(* PLC project Template, CODESYS CODESYS V3.5 SP17 Patch 3 *)
(* stored: creationDateTime 2026-02-13T14:33:38.6413633, version 3.5.17.30, modificationDateTime 2026-02-13T14:07:44.0721923, organization organization *)

{attribute 'qualified_only'}
{attribute 'strict'}
TYPE e_SaveReadJSONFileStates : (STATE_IDLE := 0, STATE_COMBINE, STATE_COMPOSE, STATE_SAVE, STATE_FINISH, STATE_PARSE, STATE_READ);
END_TYPE

FUNCTION_BLOCK FB_ReadJSONFile
  VAR CONSTANT
    SplitSize : INT := 1024;
  END_VAR
  VAR_INPUT
    xStart : BOOL;
    sFileName : STRING(255);
    pJSOBJ : POINTER TO ARRAY[1..GPL_JSON.MAX_VARS] OF JSONVAR;  (* pointer to local structure made up of type JSONVAR *)
    udiSize : UDINT;  (* SHOULD BE EQUAL TO SIZEOF(JSONOBJ) , *)
  END_VAR
  VAR_OUTPUT
    xBusy : BOOL;
    xDone : BOOL;
    xError : BOOL;
  END_VAR
  VAR
    state : e_SaveReadJSONFileStates := e_SaveReadJSONFileStates.STATE_IDLE;
    xStartRE : R_TRIG;
    xAutoReset : BOOL := TRUE;
    fread : FB_ReadTxtFile;
    ParseJSON : JSON_TO_STRUCT;  (* Part of PRO_JSON *)
    sContent : STRING(GPL_JSON.MAX_JSON_STRING);
    sLastError : STRING;
  END_VAR

            xStartRE(CLK:=xStart);
CASE state OF
	e_SaveReadJSONFileStates.STATE_IDLE:
		IF xStartRE.Q THEN
			state:=e_SaveReadJSONFileStates.STATE_READ;
			xDone:=FALSE;
			xBusy:=TRUE;
			xError:=FALSE;
			sLastError:='';
			sContent:='';
		END_IF

	e_SaveReadJSONFileStates.STATE_READ:
		fread(sFileName:=sFileName,
			result:=sContent,
			xStart:=TRUE);	
	
		IF fread.xDone THEN
			state:=e_SaveReadJSONFileStates.STATE_PARSE;
		END_IF
		IF fread.xError THEN
			state:=e_SaveReadJSONFileStates.STATE_FINISH;
			xError:=TRUE;
			sLastError:='File reading';
		END_IF

	e_SaveReadJSONFileStates.STATE_PARSE:
		ParseJSON(JSONString:=ADR(sContent),
				JSONStringSize:=SIZEOF(sContent),
				JSONVars:=pJSOBJ,
				NumberOfVars:=udiSIZE/SIZEOF(JSONVAR),
				Execute:=TRUE);

		IF  ParseJSON.Done THEN
			state:=e_SaveReadJSONFileStates.STATE_FINISH;
		END_IF
		IF ParseJSON.Error THEN
			state:=e_SaveReadJSONFileStates.STATE_FINISH;
			xError:=TRUE;
			sLastError:='JSON parsing';
		END_IF

	e_SaveReadJSONFileStates.STATE_FINISH:
		xBusy:=FALSE;
		xDone:=TRUE;

		IF xAutoReset THEN
			Reset();
		END_IF
		ParseJSON(Execute:=TRUE);
		state:=e_SaveReadJSONFileStates.STATE_IDLE;
END_CASE

          

METHOD Reset : BOOL
                  state:=e_SaveReadJSONFileStates.STATE_IDLE;
sContent:='';
ParseJSON(Execute:=FALSE);
ParseJSON.ClearAll();
xError:=FALSE;
Reset:=TRUE;
xStartRE(CLK:=FALSE);
                
END_METHOD
END_FUNCTION_BLOCK

{attribute 'contains_implicit_enum'}
FUNCTION_BLOCK FB_ReadTxtFile
  VAR CONSTANT
    SplitSize : INT := 1024;
  END_VAR
  VAR_INPUT
    xStart : BOOL;
    sFileName : REFERENCE TO STRING(255);
    Result : REFERENCE TO STRING(GPL_JSON.MAX_JSON_STRING);
  END_VAR
  VAR_OUTPUT
    xBusy : BOOL;
    xDone : BOOL;
    xError : BOOL;
  END_VAR
  VAR
    fopen : FILE.Open;
    fread : FILE.Read;
    fclose : FILE.Close;
    xStartRE : R_TRIG;
    xAutoReset : BOOL := TRUE;
    {attribute 'implicit_enum_type'}
    step : Implicit_Enum__FB_ReadTxtFile__step;
    tempString : STRING(GPL_JSON.MAX_JSON_STRING);
    endPos : INT;
    subString : STRING(SplitSize);  (* Not more than CLEANSTRING.MAXSTRING; *)
    cleanupCount : INT := 0;
    cleanupCounter : INT;
    tmp : REAL;
    startPos : INT;
    finishPos : INT;
    lenCopy : DINT;
    pos : INT;
    testChar : STRING(1) := '"';
    testStr : STRING(1);
  END_VAR

            xStartRE(CLK:=xStart);
CASE step OF
	STEP_IDLE:
		IF xStartRE.Q AND NOT xError THEN
			step:=STEP_OPEN;
			xDone:=FALSE;
			xBusy:=TRUE;
			xError:=FALSE;			
		END_IF
		
		fopen(xExecute:=FALSE);
    	fread(xExecute:=FALSE);
		fclose(xExecute:=FALSE);
	
	STEP_OPEN:
		fopen.sFileName:=sFileName;
		fopen.eFileMode:=FILE.MODE.MREAD;
		fopen.xExclusive:=TRUE;
		fopen(xExecute:=TRUE);
		
		IF fopen.xDone THEN
			step:=STEP_READ;
		END_IF
		IF fopen.xError THEN
			step:=STEP_CLOSE;
			xError:=TRUE;
		END_IF
		
	STEP_READ:
		Result:='';
		fread.hFile:=fopen.hFile;
		
		fread.pBuffer:=ADR(tempString);
		
		fread.szBuffer:=SIZEOF(tempString);
		fread(xExecute:=TRUE);
		IF fread.xDone THEN
			step:=STEP_CLEANUP;
			endPos:=TO_INT(StrLenA(ADR(tempString)));
			startPos:=1; 
			cleanupCounter:=0;
			
			cleanupCount:=TO_INT(endPos/SplitSize);
			//Simple Round up
			tmp:=TO_REAL(endPos)/TO_REAL(SplitSize);
			IF tmp>TO_REAL(cleanupCount) THEN
				cleanupCount:=cleanupCount+1;
			END_IF
			
		END_IF
		IF fread.xError THEN
			step:=STEP_CLOSE;
			xError:=TRUE;
		END_IF
	STEP_CLEANUP:
		
		finishPos := MIN(endPos, startPos + SplitSize - 1);
		pos:=finishPos;
		lenCopy   := finishPos - startPos + 1;  
		IF lenCopy>0 THEN
			STU.StrMidA(ADR(tempString),SIZEOF(tempString),TO_INT(lenCopy),startPos,ADR(subString),TO_UINT(SplitSize+1));
			CleanupString(); //Save spaces
			STU.StrConcatA(ADR(subString),ADR(Result),TO_INT(SIZEOF(Result)));
		END_IF
		
		IF finishPos>=endPos THEN 
			step:=STEP_CLOSE;
		END_IF
		startPos:=finishPos+1;
		cleanupCounter:=cleanupCounter+1;
		IF cleanupCounter>cleanupCount THEN 
			step:=STEP_CLOSE;
		END_IF
	STEP_CLOSE:
		fclose.hFile:=fopen.hFile;
		fclose(xExecute:=TRUE);
		IF fclose.xDone THEN
			step:=STEP_FINISH;
		END_IF
		IF fclose.xError THEN
			step:=STEP_FINISH;
			xError:=TRUE;
		END_IF
		
	STEP_FINISH:
		IF xAutoReset AND xError THEN
			Reset();
		END_IF
		step:=STEP_IDLE;
		xDone:=TRUE;
		xStart:=FALSE;
		xBusy:=FALSE;
END_CASE
          

METHOD Reset : BOOL
                  xStartRE(CLK:=FALSE);
xError:=FALSE;
                
END_METHOD

(* | | Edit: allow for space symol | | Original: | | Author: Tim Van Meppelen, Pro Electric Inc. | timv@proelectric.com | Date: Oct 9, 2018 | strip all control characters and spaces from a string EXCEPT space *)
METHOD CleanupString : BOOL
  VAR
    StringPtr : POINTER TO ARRAY[1..GPL_JSON.MAX_JSON_STRING] OF ASCII;
    i : UINT;
    j : UINT;
  END_VAR
                  StringPtr:=ADR(THIS^.subString);
FOR i:= 1 TO GPL_JSON.MAX_JSON_STRING DO
	//IF (StringPtr^[i] >= 1) AND (StringPtr^[i] <= 16#20) THEN
	IF (StringPtr^[i] >= 1) AND (StringPtr^[i] < 16#20) THEN
	//match all control and white space characters, except for null AND SPACE, which terminates a string
		FOR j:= i TO GPL_JSON.MAX_JSON_STRING DO
			IF (StringPtr^[j] = PRO_JSON.ASCII.NULL) THEN
			//null character terminates string
				EXIT;
			ELSE
			//shift character array left one
				StringPtr^[j]:= StringPtr^[j+1];
			END_IF
		END_FOR
		i:= i - 1;	//run loop at same position again
	ELSIF (StringPtr^[i] = PRO_JSON.ASCII.NULL) THEN
	//found null character at the end of the string
		EXIT;
	END_IF
END_FOR

CleanupString:= TRUE;

                
END_METHOD
END_FUNCTION_BLOCK

FUNCTION_BLOCK FB_SaveJSONFile
  VAR_INPUT
    xStart : BOOL;
    sFileName : STRING(255);
    pJSOBJ : POINTER TO ARRAY[1..GPL_JSON.MAX_VARS] OF JSONVAR;  (* pointer to local structure made up of type JSONVAR *)
    udiSize : UDINT;  (* SHOULD BE EQUAL TO SIZEOF(JSONOBJ) , //JSONVAR is part of JSON lib *)
    IgnoreNull : BOOL := FALSE;  (* Ignore null objects when exporting (Default: False, do not ignore) *)
    Format : BOOL := TRUE;  (* Format JSON when expoting with Tabs and newlines (Default: True, format it. Format values are library parameters) *)
    CustomFieldName : STRING(GPL_JSON.MAX_VAR_NAME);  (* Name of optional custom field, that will be added to the end of the root *)
    pCustomFieldString : POINTER TO STRING(GPL_JSON.MAX_JSON_STRING);  (* Pointer to long custom string. *)
  END_VAR
  VAR_OUTPUT
    xBusy : BOOL;
    xDone : BOOL;
    xError : BOOL;
  END_VAR
  VAR
    state : e_SaveReadJSONFileStates := e_SaveReadJSONFileStates.STATE_IDLE;
    xAutoReset : BOOL := TRUE;
    xStartRE : R_TRIG;
    fsave : FB_SaveTxtFile;  (* Other FB *)
    ComposeJSON : STRUCT_TO_JSON;  (* STRUCT_TO_JSON FB is part of JSON lib *)
    sContent : STRING(GPL_JSON.MAX_JSON_STRING);
    sLastError : STRING;
    sNote : STRING := 'I AM NOTE';
  END_VAR

            xStartRE(CLK:=xStart);
CASE state OF
	e_SaveReadJSONFileStates.STATE_IDLE:
		IF xStartRE.Q THEN
			state:=e_SaveReadJSONFileStates.STATE_COMPOSE;
			xDone:=FALSE;
			xBusy:=TRUE;
			xError:=FALSE;
			sLastError:='';
			sContent:='';
		END_IF

	e_SaveReadJSONFileStates.STATE_COMPOSE:
		IF LEN(CustomFieldName)>0 AND StrLenA(pCustomFieldString)>0 THEN 
			ComposeJSON.SetCustomField(Name:=CustomFieldName,TextPtr:=pCustomFieldString);
		END_IF
		ComposeJSON(
			JSONString:= ADR(sContent),
			JSONStringSize:= SIZEOF(sContent),
			JSONVars:= pJSOBJ,
			NumberOfVars:= udiSize / SIZEOF(JSONVAR), //JSONVAR is part of JSON lib
			Execute:=TRUE,
			IgnoreNull:=IgnoreNull,
			Format:=Format
		);

		IF ComposeJSON.Done THEN
			state:=e_SaveReadJSONFileStates.STATE_SAVE;
		END_IF
		IF ComposeJSON.Error THEN
			state:=e_SaveReadJSONFileStates.STATE_FINISH;
			xError:=TRUE;
			sLastError:='JSON Composing';
		END_IF

	e_SaveReadJSONFileStates.STATE_SAVE:
		fsave.sContent REF=sContent;
		fsave.sFileName REF=sFileName;

		fsave(xStart:=TRUE);

		IF  fsave.xDone THEN
			state:=e_SaveReadJSONFileStates.STATE_FINISH;
		END_IF
		IF fsave.xError THEN
			state:=e_SaveReadJSONFileStates.STATE_FINISH;
			xError:=TRUE;
			sLastError:='File saving';
		END_IF

	e_SaveReadJSONFileStates.STATE_FINISH:
		xBusy:=FALSE;
		xDone:=TRUE;

		IF xAutoReset THEN
			Reset();
		END_IF
		
		state:=e_SaveReadJSONFileStates.STATE_IDLE;
END_CASE

          

METHOD Reset : BOOL
                  state:=e_SaveReadJSONFileStates.STATE_IDLE;
xStartRE(CLK:=FALSE);
sContent:='';
ComposeJSON(Execute:=FALSE);
ComposeJSON.ClearString();

xError:=FALSE;


Reset:=TRUE;
                
END_METHOD
END_FUNCTION_BLOCK

{attribute 'contains_implicit_enum'}
FUNCTION_BLOCK FB_SaveTxtFile
  VAR CONSTANT
    SplitSize : INT := 1024;
  END_VAR
  VAR_INPUT
    xStart : BOOL;
    sFileName : REFERENCE TO STRING(255);
    sContent : REFERENCE TO STRING(GPL_JSON.MAX_JSON_STRING);
  END_VAR
  VAR_OUTPUT
    xBusy : BOOL;
    xDone : BOOL;
    xError : BOOL;
  END_VAR
  VAR
    fopen : FILE.Open;
    fwrite : FILE.Write;
    fclose : FILE.Close;
    {attribute 'implicit_enum_type'}
    step : Implicit_Enum__FB_SaveTxtFile__step;
    xStartRE : R_TRIG;
    xAutoReset : BOOL := TRUE;
  END_VAR

            xStartRE(CLK:=xStart);
CASE step OF
	STATE_IDLE:
		IF xStartRE.Q AND NOT xError THEN
			step:=STATE_OPEN;
			xDone:=FALSE;
			xBusy:=TRUE;
			xError:=FALSE;			
		END_IF
		fopen(xExecute:=FALSE);
    	fwrite(xExecute:=FALSE);
		fclose(xExecute:=FALSE);

	STATE_OPEN:
		fopen.sFileName:=sFileName;
		fopen.eFileMode:=FILE.MODE.MWRITE;
		fopen.xExclusive:=TRUE;
		fopen(xExecute:=TRUE);
		IF fopen.xDone THEN
			step:=STATE_WRITE;
		END_IF
		IF fopen.xError THEN
			step:=STATE_CLOSE;
			xError:=TRUE;
		END_IF

	STATE_WRITE:
		fwrite.hFile:=fopen.hFile;
		fwrite.pBuffer:=ADR(sContent);
		fwrite.szSize:=TO___UXINT(STU.StrLenA(ADR(sContent)));
		fwrite(xExecute:=TRUE);		
		IF fWrite.xDone THEN
			step:=STATE_CLOSE;
		END_IF
		IF fWrite.xError THEN
			step:=STATE_CLOSE;
			xError:=TRUE;
		END_IF
		
	STATE_CLOSE:
		fclose.hFile:=fopen.hFile;
		fclose(xExecute:=TRUE);
		IF fclose.xDone THEN
			step:=STEP_FINISH;
		END_IF
		IF fclose.xError THEN
			step:=STEP_FINISH;
			xError:=TRUE;
		END_IF
		
	STEP_FINISH:
		IF xAutoReset THEN
			Reset();
		END_IF
		step:=STATE_IDLE;
		xDone:=TRUE;
		xStart:=FALSE;
		xBusy:=FALSE;

END_CASE
          

METHOD Reset : BOOL
                  xError:=FALSE;
step:=STATE_IDLE;

xStartRE(CLK:=FALSE);
                
END_METHOD
END_FUNCTION_BLOCK
